PROGRAM main
VAR
	InputA AT %IX0.1 : bool;
	InputB AT %IX0.2 : bool;
	Output AT %QX0.0 : bool;
	Input : bool;
END_VAR

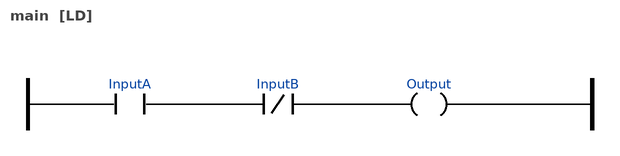
(* LD diagram, written out as Structured Text *)
Output := InputA AND NOT InputB;
END_PROGRAM
